PROGRAM MAIN
VAR
	xBool	: BOOL;
	xSigC	AT %I* : BOOL;
	xSigO	AT %I* : BOOL;
	iHumidityRaw AT %I* : INT;
	iTempRaw	AT %I* : INT;
	fbTONR	: TONReset;
END_VAR

fbTONR(PT	:= T#4S);

IF fbTONR.rtTimerDone.Q THEN
	xBool	:= TRUE;
END_IF

END_PROGRAM

(* stored: Version 1.1.0.1, ProductVersion 3.1.4024.9
   POU MAIN: Id {e5d15e63-e8ca-4ab2-8b70-a028e7480ab2}, SpecialFunc None *)
